FUNCTION_BLOCK Constanzia_Object EXTENDS TcoCore.TcoObject
VAR
    _victor : AKid_Object(THIS^);
    _michael : AKid_Object(THIS^);
END_VAR

END_FUNCTION_BLOCK

(* stored: Version 1.1.0.1, ProductVersion 3.1.4024.9
   POU Constanzia_Object: Id {2054403e-1d36-0b1d-3ac2-42531aa5b0ec}, SpecialFunc None *)
